(* IEC 61131-3 sources: AXOpen/src/abstractions/ctrl/src/AxoMessenger, 3 files *)

(* ---- IAxoMessenger.st ---- *)
NAMESPACE AXOpen.Core
    INTERFACE PUBLIC IAxoMessenger

    END_INTERFACE
END_NAMESPACE

(* ---- IAxoMessengerService.st ---- *)
NAMESPACE AXOpen.Core
     INTERFACE PUBLIC IAxoMessagingServices
        METHOD QueueMessage : BOOL
             VAR_INPUT
                inMessegenger : IAxoMessenger;
            END_VAR
        END_METHOD
        /// <summary>
        /// Suspends the messaging system. When suspended, messages will not be sent to subscribers until the system is resumed.
        /// This is useful for scenarios where you want to temporarily prevent messages from being processed.
        /// </summary>
        METHOD SuspendMessaging END_METHOD

        /// <summary>
        /// Resumes the messaging system. When resumed, messages that arose while the system was suspended will NOT be sent to subscribers.
        /// </summary>
        METHOD ResumeMessaging END_METHOD

        /// <summary>
        /// Checks if the messaging system is currently suspended.
        /// Returns true if the messaging system is suspended, false otherwise.
        /// </summary>
        METHOD IsSuspended : BOOL END_METHOD

        /// <summary>
        /// Requalifies the message category for downstream messages.
        /// This is used to ensure that messages that are sent from a downstream component are categorized correctly,
        /// even if the upstream component has a different message category.
        /// </summary>
        METHOD RequalifyDownstreamMessages
            VAR_INPUT
                inMessageCategory : AXOpen.Messaging.eAxoMessageCategory;
            END_VAR
        END_METHOD

        /// <summary>
        /// Gets the requalified message category for downstream messages.
        /// </summary>
        METHOD GetRequalifiedMessageCategory : AXOpen.Messaging.eAxoMessageCategory END_METHOD
    END_INTERFACE
END_NAMESPACE

(* ---- eAxoMessageCategory.st ---- *)
NAMESPACE AXOpen.Messaging
    TYPE PUBLIC
        ///<summary>
        /// Message categories.
        /// ATTENTION: Values must be multiply of 100
        ///</summary>
        eAxoMessageCategory : INT
        (
            ///<summary>
            /// No category.
            /// This is used to indicate that the message does not have any importance and should be ignored by the system.
            /// Do not use this category for messages that have to be delivered to the user, even if such information is not critical.
            /// </summary>
            None := 0,

            ///<summary>
            /// Info message.
            /// Use when you want to deliver information to the user, that has only informative character and does not adversely affect a process.
            ///</summary>
            Info := 100,

            ///<summary>
            /// Potential problem message.
            /// Use this category when you want to report to the user an information about a potential problem, that does not necessarily affect a process
            /// but may cause a problem. This is typically used when certain conditions is expected to happen within a process that did not happen yet,
            /// this category is aimed to be later automatically requalified to Warning or Error by coordination primitive if the expected conditions did not happen within expected time.
            ///</summary>
            Potential := 150,

            ///<summary>
            /// Warning message.
            /// Use this category when you want to report to the user an information about a possible problem, that may adversly affect a process.
            /// Information in this cateogory aims to help the user to identify a problem, the cause of such problem does not necessarily stops the process.
            ///</summary>
            Warning := 200,

            ///<summary>
            /// Error message.
            /// Use this category when there is a failure that cannot be immediately recovered and an intervention is needed. This is typically a situation when a device fails
            /// to deliver expected result.
            /// Do not use this category to report information about failed process like measurement or detection.
            ///</summary>
            Error := 300,

            ///<summary>
            /// Programming error.
            /// Use this category to report programming errors, like invalid parameters, invalid state of the object etc.
            ///</summary>
            ProgrammingError := 400,

            ///<summary>
            /// Critical error.
            /// Use this category when a critical error occured, that is not recoverable by the means of software (reset/restore) but device still operates under such conditions; a detailed inspection and an expert action is required.
            ///</summary>
            Critical := 500
        );
    END_TYPE
END_NAMESPACE
